(* PLC project Unnamed, Unknown Unnamed 1 *)
(* stored: creationDateTime 2020-09-15T10:36:20, modificationDateTime 2025-06-04T19:27:11 *)

PROGRAM part1c
  VAR
    Input0 AT %IX1.0 : BOOL;
    Output0 AT %QX1.0 : BOOL;
  END_VAR
  VAR
    Oscillator : BOOL;
    TON0 : TON;
    TOF0 : TOF;
    TON1 : TON;
    CTU0 : CTU;
  END_VAR
  VAR  (* added by the conversion: wires and edge detectors of the diagram *)
    R_TRIG1 : R_TRIG;
    R_TRIG2 : R_TRIG;
  END_VAR

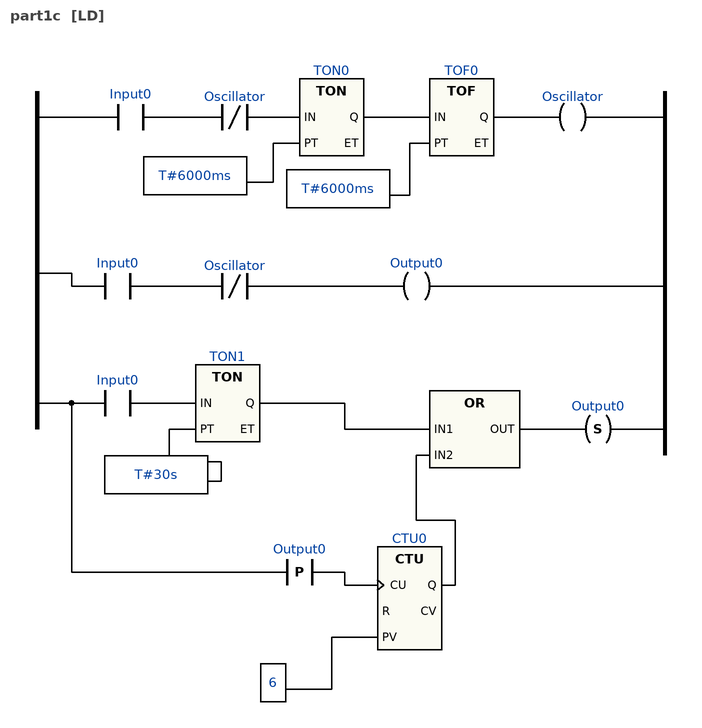
(* LD diagram, written out as Structured Text *)
TON0(IN := Input0 AND NOT Oscillator, PT := T#6000ms);
TOF0(IN := TON0.Q, PT := T#6000ms);
Oscillator := TOF0.Q;
Output0 := Input0 AND NOT Oscillator;
TON1(IN := Input0, PT := T#30s);
R_TRIG1(CLK := Output0);
R_TRIG2(CLK := R_TRIG1.Q);
CTU0(CU := R_TRIG2.Q, PV := 6);
IF TON1.Q OR CTU0.Q THEN Output0 := TRUE; END_IF;
END_PROGRAM

CONFIGURATION Config0
  RESOURCE Res0 ON PLC
    TASK task0(INTERVAL := T#20ms, PRIORITY := 0);
    PROGRAM instance0 WITH task0 : part1c;
  END_RESOURCE
END_CONFIGURATION
